PROGRAM MAIN
VAR
END_VAR

END_PROGRAM

(* stored: Version 1.1.0.1
   POU MAIN: Id {28360960-9ab2-43c1-b11c-05f0dfab6dbb} *)
